// TIA Portal V21 export
TYPE "LAxisCtrl_typeGearInRelative"
TITLE = LAxisCtrl_typeGearInRelative
// Support: tech.team.motioncontrol@siemens.com
   STRUCT
      ratioNumerator : DInt := 1;   // Gear ratio numerator (permitted integer values: -2147483648 to 2147483647; value 0 not permitted)
      ratioDenominator : DInt := 1;   // Gear ratio denominator (permitted integer values: 1 to 2147483647)
      acceleration : LReal := -1.0;   // Acceleration for synchronization (Value > 0.0: The specified value is used; Value = 0.0: Not permitted; Value < 0.0: Use of the default value configured in the technology object)
      deceleration : LReal := -1.0;   // Deceleration for synchronization (Value > 0.0: The specified value is used; Value = 0.0: Not permitted; Value < 0.0: Use of the default value configured in the technology object)
      jerk : LReal := -1.0;   // Jerk for synchronization (Value > 0.0: Smooth velocity profile, the specified value is used; Value = 0.0: Trapezoid velocity profile; Value < 0.0: Use of the default value configured in the technology object)
      ratioChangeOnTheFly : Bool := FALSE;   // TRUE: Changing gear ratio on-the-fly; FALSE: Ratio change requires a new rising edge at gearInRelative input
   END_STRUCT;
END_TYPE
